ABB RobotStudio station: assigment 2.rsstn

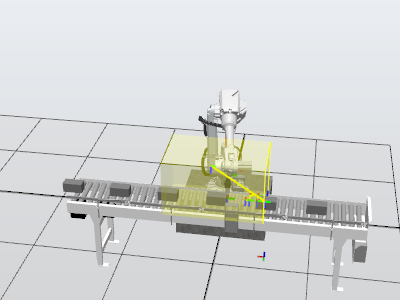
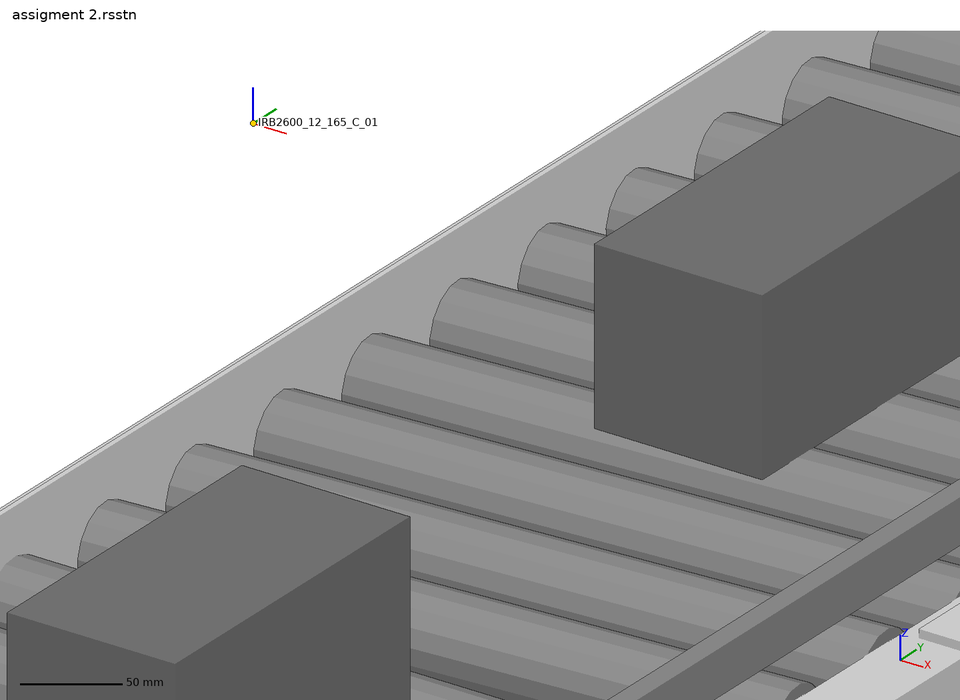
[picture v1: parts stored in the station drawn from their meshes, with robot base, taught points and paths (robot models come from the ABB library and are not in the file)]
Station Station (saved by RobotStudio 22.3.10141.1)
Controller Controller10, task T_ROB1: task frame (RAPID world) sits at (798.13, 524.53, 0) mm, rotated rx 0 ry 0 rz -89.92 deg in the station
Controller Controller10
  mechanical unit ROB_1: IRB2600_12_165_C_01, 6 joints, base frame (523.48, -798.82, 245.81) mm, rotated rx 0 ry 0 rz 89.92 deg
  mechanical unit CNV1: ?, 1 joints, base frame (0, 2.5, 775) mm
Layout (positions relative to the parent item):
  - Concrete [part, from Dispencing\Concrete.rslib]
  - IRB2600_12_165_C_01 [mechanism, from %ABB.RobotStudio.Models.IRB2600%\IRB2600_12_165_C_01.rslib] at (0, 0, 245.8) mm; joint values [0.1622, -0.034, 0.4957, -0.2395, 0.4438, 0.3433] (rad or m)
  - MyTool [mechanism, from Training Objects\myTool.rslib] at (931.18, 143.56, 1073.22) mm, rotated rx -180 ry 39.12 rz -180 deg
  - Conveyor [conveyor]
    - 400_guide [part] at (796.82, 1524.53, 0) mm, rotated rx 0 ry 0 rz -89.92 deg, size 3033 x 590 x 945 mm
    - Part_1 [part], size 200 x 100 x 100 mm
    - ConveyorObject_21 [conveyorobject] at (803.13, -1371.11, 775) mm, rotated rx 0 ry 0 rz -89.92 deg
      - Part_1 [part] at (0, 150, 0) mm, size 200 x 100 x 100 mm
    - ConveyorObject_22 [conveyorobject] at (802.47, -871.11, 775) mm, rotated rx 0 ry 0 rz -89.92 deg
      - Part_1 [part] at (0, 150, 0) mm, size 200 x 100 x 100 mm
    - ConveyorObject_23 [conveyorobject] at (801.81, -371.11, 775) mm, rotated rx 0 ry 0 rz -89.92 deg
      - Part_1 [part] at (0, 150, 0) mm, size 200 x 100 x 100 mm
    - ConveyorObject_24 [conveyorobject] at (801.15, 128.89, 775) mm, rotated rx 0 ry 0 rz -89.92 deg
      - Part_1 [part] at (0, 150, 0) mm, size 200 x 100 x 100 mm
    - ConveyorObject_25 [conveyorobject] at (800.5, 628.89, 775) mm, rotated rx 0 ry 0 rz -89.92 deg
      - Part_1 [part] at (0, 150, 0) mm, size 200 x 100 x 100 mm
    - ConveyorObject_26 [conveyorobject] at (799.84, 1128.89, 775) mm, rotated rx 0 ry 0 rz -89.92 deg
      - Part_1 [part] at (0, 150, 0) mm, size 200 x 100 x 100 mm
Attachment: MyTool is attached to IRB2600_12_165_C_01 / Link6
Conveyor tracking Connection: unit CNV1, TravelOffset=0.925156, QueueTrackDistance=0, StartWindowWidth=1, SyncSeparation=0.1, CountsPerMeter=10000
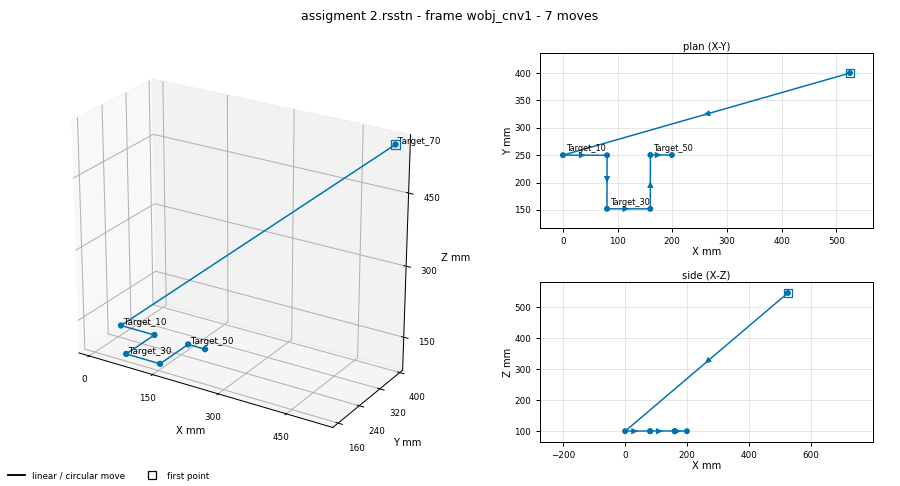
[picture p0: tool path of assigment 2.rsstn in frame wobj_cnv1, 7 of 7 moves have a stored position in this frame; points joined in program order, loops and branches not executed]
Targets, tools, work objects and paths stored in the station, written as RAPID:
! task T_ROB1
MODULE CalibData
  PERS tooldata MyTool:=[TRUE,[[31.792631019,0,229.638935148],[0.945518576,0,0.325568154,0]],[1,[0,0,1],[1,0,0,0],0,0,0]];
  TASK PERS wobjdata wobj_cnv1:=[FALSE,FALSE,"CNV1",[[0,0,0],[1,0,0,0]],[[0,0,0],[1,0,0,0]]];
ENDMODULE

! task T_ROB1
MODULE Module1
  CONST robtarget Target_10:=[[0.000009635,250.000343469,99.999971032],[0.006922145,-0.706607065,0.707538515,0.006913002],[0,-1,0,0],[9E+09,9E+09,9E+09,9E+09,9E+09,0]];
  CONST robtarget Target_20:=[[80.648820828,249.894109754,99.999974431],[0.006922099,-0.706607065,0.707538515,0.006912966],[0,-1,0,0],[9E+09,9E+09,9E+09,9E+09,9E+09,0]];
  CONST robtarget Target_30:=[[80.519699626,151.890070359,99.999964724],[0.006922065,-0.706607073,0.707538508,0.006912908],[0,-1,0,0],[9E+09,9E+09,9E+09,9E+09,9E+09,0]];
  CONST robtarget Target_40:=[[159.76152419,151.785691254,99.999982965],[0.00692202,-0.706607076,0.707538506,0.006912875],[0,-1,0,0],[9E+09,9E+09,9E+09,9E+09,9E+09,0]];
  CONST robtarget Target_50:=[[159.891335367,250.321741519,99.999984971],[0.006921981,-0.706607077,0.707538506,0.006912844],[0,-1,0,0],[9E+09,9E+09,9E+09,9E+09,9E+09,0]];
  CONST robtarget Target_60:=[[199.272226523,250.26986095,99.999981151],[0.006921933,-0.706607066,0.707538518,0.006912809],[0,-1,0,0],[9E+09,9E+09,9E+09,9E+09,9E+09,0]];
  CONST robtarget Target_70:=[[525.058527209,400.264477782,545.95188716],[0.135011179,-0.693657873,0.694572301,0.134833432],[0,0,0,0],[9E+09,9E+09,9E+09,9E+09,9E+09,0]];
  PROC Path_10()
    ActUnit CNV1;
    WaitWObj wobj_cnv1;
    MoveL Target_70,v1000,z100,MyTool\WObj:=wobj_cnv1;
    MoveL Target_10,v1000,z100,MyTool\WObj:=wobj_cnv1;
    MoveL Target_20,v1000,z100,MyTool\WObj:=wobj_cnv1;
    MoveL Target_30,v1000,z100,MyTool\WObj:=wobj_cnv1;
    MoveL Target_40,v1000,z100,MyTool\WObj:=wobj_cnv1;
    MoveL Target_50,v1000,z100,MyTool\WObj:=wobj_cnv1;
    MoveL Target_60,v1000,z100,MyTool\WObj:=wobj_cnv1;
    WaitTime 1;
    DropWObj wobj_cnv1;
  ENDPROC
ENDMODULE

